(* CoDeSys 2.3.9.37 project: Cap11_3.pro *)
(* Libraries: Standard.lib 4.10.05 12:14:46, IecSfc.lib 13.4.06 16:51:28 *)

(* POU PLC_PRG, SFC *)
PROGRAM PLC_PRG
VAR
      (* Entradas *)
	A: BOOL;
	B: BOOL;
	Inc: BOOL;
	Resetea: BOOL;
      (* Salidas *)
	Salida: BOOL;
      (* Otras *)
	MiContador: CTU;
	Valor : INT;

END_VAR
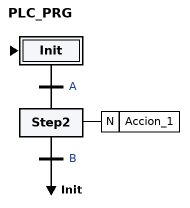
INITIAL_STEP Init:
END_STEP
TRANSITION FROM Init TO Step2 := A;
END_TRANSITION
STEP Step2:
	Accion_1(N);
END_STEP
TRANSITION FROM Step2 TO Init := B;
END_TRANSITION
END_PROGRAM
ACTION Accion_1:
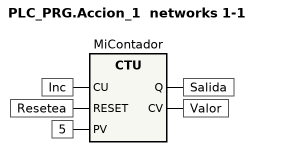
_FBD_ (* Function Block Diagram *)
NETWORK 1
	MiContador:CTU(CU: Inc, RESET: Resetea, PV: 5, CV => Valor) => Salida
_END_FBD_
(* the same logic as Structured Text *)
(* Network 1 *)
MiContador(CU := Inc, RESET := Resetea, PV := 5);
Valor := MiContador.CV;
Salida := MiContador.Q;
END_ACTION

(* Visualisation Visu
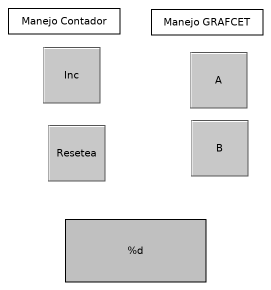
button at (80,54)-(137,110): text "Inc"; taps PLC_PRG.Inc
button at (85,132)-(142,188): text "Resetea"; taps PLC_PRG.Resetea
button at (227,59)-(284,115): text "A"; taps PLC_PRG.A
button at (228,127)-(285,183): text "B"; taps PLC_PRG.B
rectangle at (45,15)-(157,41): text "Manejo Contador"
rectangle at (188,16)-(300,42): text "Manejo GRAFCET"
rounded rectangle at (102,226)-(243,289): text "%d"; shows PLC_PRG.MiContador.CV; alarm colour if PLC_PRG.Salida
*)
